PROGRAM MAIN
VAR
	MyVar AT%I*:UDINT;
	StatusWordDrive2 AT%I*:UINT;
END_VAR

END_PROGRAM

(* stored: Version 1.1.0.1, ProductVersion 3.1.4024.10
   POU MAIN: Id {500e18b9-5408-4d9f-adda-d2a5f4f3009f}, SpecialFunc None *)
